PROGRAM TEST_MAIN
VAR
	clientConnectionTest 	: FB_OPCUA_ClientConnection_Test;
	workOnNodeTest			: FB_OPCUA_WorkOnNode_Test;
	startTest: BOOL;
	testBool : BOOL;
	value: usint;
	cbData: UDINT;
		opcUAreadList_BOOL: ST_OPCUA_NodeVariablePair_BOOL := (clientvariable := testBool, 
															serverNodeIdentifier := 'booleantoread'//,
															);//clientVariableInfo := __VARINFO(THIS^.opcUAreadList_BOOL));
	testADd : PVOID;
	testInfo : __SYSTEM.VAR_INFO;
	
	var1 : STRING;
	var2 : BYTE;
	add1 : PVOID;
	add2 : PVOID;
	
	clientVarInfo : __SYSTEM.VAR_INFO;
	clientByteValue : BYTE;
	pt : POINTER TO BYTE;
	
END_VAR

IF startTest THEN
	TcUnit.RUN();
END_IF

END_PROGRAM

(* stored: Version 1.1.0.1, ProductVersion 3.1.4024.9
   POU TEST_MAIN: Id {6f1f9b14-cd50-4368-a31b-0aa59c1c9cf4}, SpecialFunc None *)
